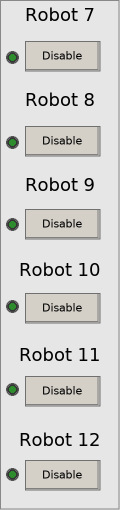
VISUALIZATION RightRobotControls  // 120x510
    Textfield (0,0 120x30), "Robot 7"
    Textfield (0,85 120x30), "Robot 8"
    Textfield (0,170 120x30), "Robot 9"
    Textfield (0,255 120x30), "Robot 10"
    Textfield (0,340 120x30), "Robot 11"
    Textfield (0,425 120x30), "Robot 12"
    Button (25,41 75x30), "Disable"
    Button (25,126 75x30), "Disable"
    Button (25,209 75x30), "Disable"
    Button (25,293 75x30), "Disable"
    Button (25,376 75x30), "Disable"
    Button (25,460 75x30), "Disable"
    Lamp1 (5,50 15x15), variable: TRUE, style: Lamp-Lamp1-Green
    Lamp1 (5,135 15x15), variable: TRUE, style: Lamp-Lamp1-Green
    Lamp1 (5,217 15x15), variable: TRUE, style: Lamp-Lamp1-Green
    Lamp1 (5,299 15x15), variable: TRUE, style: Lamp-Lamp1-Green
    Lamp1 (5,382 15x15), variable: TRUE, style: Lamp-Lamp1-Green
    Lamp1 (5,467 15x15), variable: TRUE, style: Lamp-Lamp1-Green
END_VISUALIZATION

(* stored: Version 1.1.0.1, ProductVersion 3.1.4024.15
   Visu RightRobotControls: Id {542f153f-f835-4bef-b474-855b9d7f2705} *)
